Omron CX-Programmer project NewProject (CX-Programmer 9.61)

# PLC NewPLC1: CP1E E20

## Global symbols (name address type ; comment)
0.12 BOOL  ; StopButton
10.00 BOOL  ; Conveyor
0.04 BOOL  ; BothSW
0.03 BOOL  ; BlueSW
0.02 BOOL  ; YellowSW
0.00 BOOL  ; StartButton
0.01 BOOL  ; JobINSen
0.05 BOOL  ; YTHLS
0.06 BOOL  ; BTHLS
0.07 BOOL  ; YTLLS
0.08 BOOL  ; BTLLS
0.09 BOOL  ; JobOUTSen
0.10 BOOL  ; FS1
0.11 BOOL  ; FS2
100.00 BOOL  ; M0
100.01 BOOL  ; M1
100.02 BOOL  ; M2
100.03 BOOL  ; M3
100.04 BOOL  ; M4
100.05 BOOL  ; M5
100.06 BOOL  ; M6
10.01 BOOL  ; YLIndicator
10.02 BOOL  ; BLIndicator
10.03 BOOL  ; YellowValve
10.04 BOOL  ; BlueValve
T000 BOOL  ; Tim1
T001 BOOL  ; Tim2
T002 BOOL  ; Tim3
T003 BOOL  ; Tim4
T004 BOOL  ; Tim5

## Program NewProgram1 (cyclic task 0)

### Section Section1

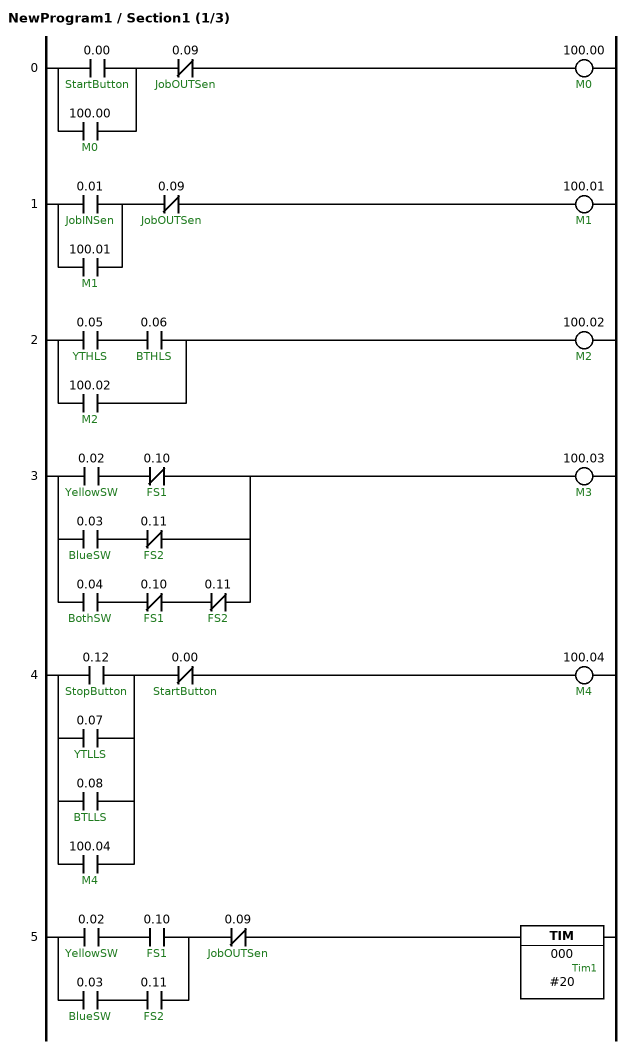
; rung 0
LD 0.00  ; StartButton
OR 100.00  ; M0
ANDNOT 0.09  ; JobOUTSen
OUT 100.00  ; M0
; rung 1
LD 0.01  ; JobINSen
OR 100.01  ; M1
ANDNOT 0.09  ; JobOUTSen
OUT 100.01  ; M1
; rung 2
LD 0.05  ; YTHLS
AND 0.06  ; BTHLS
OR 100.02  ; M2
OUT 100.02  ; M2
; rung 3
LD 0.02  ; YellowSW
ANDNOT 0.10  ; FS1
LD 0.03  ; BlueSW
ANDNOT 0.11  ; FS2
ORLD
LD 0.04  ; BothSW
ANDNOT 0.10  ; FS1
ANDNOT 0.11  ; FS2
ORLD
OUT 100.03  ; M3
; rung 4
LD 0.12  ; StopButton
OR 0.07  ; YTLLS
OR 0.08  ; BTLLS
OR 100.04  ; M4
ANDNOT 0.00  ; StartButton
OUT 100.04  ; M4
; rung 5
LD 0.02  ; YellowSW
AND 0.10  ; FS1
LD 0.03  ; BlueSW
AND 0.11  ; FS2
ORLD
ANDNOT 0.09  ; JobOUTSen
TIM 000 #20  ; Tim1

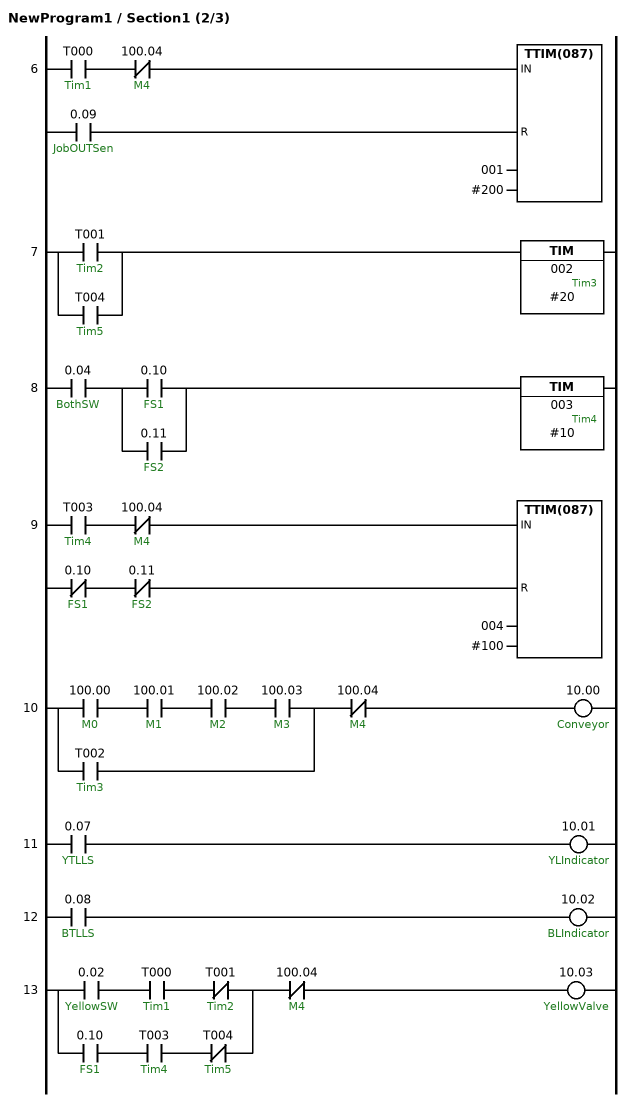
; rung 6
LD T000  ; Tim1
ANDNOT 100.04  ; M4
LD 0.09  ; JobOUTSen
TTIM(087) 001 #200  ; Tim2
; rung 7
LD T001  ; Tim2
OR T004  ; Tim5
TIM 002 #20  ; Tim3
; rung 8
LD 0.04  ; BothSW
LD 0.10  ; FS1
OR 0.11  ; FS2
ANDLD
TIM 003 #10  ; Tim4
; rung 9
LD T003  ; Tim4
ANDNOT 100.04  ; M4
LDNOT 0.10  ; FS1
ANDNOT 0.11  ; FS2
TTIM(087) 004 #100  ; Tim5
; rung 10
LD 100.00  ; M0
AND 100.01  ; M1
AND 100.02  ; M2
AND 100.03  ; M3
OR T002  ; Tim3
ANDNOT 100.04  ; M4
OUT 10.00  ; Conveyor
; rung 11
LD 0.07  ; YTLLS
OUT 10.01  ; YLIndicator
; rung 12
LD 0.08  ; BTLLS
OUT 10.02  ; BLIndicator
; rung 13
LD 0.02  ; YellowSW
AND T000  ; Tim1
ANDNOT T001  ; Tim2
LD 0.10  ; FS1
AND T003  ; Tim4
ANDNOT T004  ; Tim5
ORLD
ANDNOT 100.04  ; M4
OUT 10.03  ; YellowValve

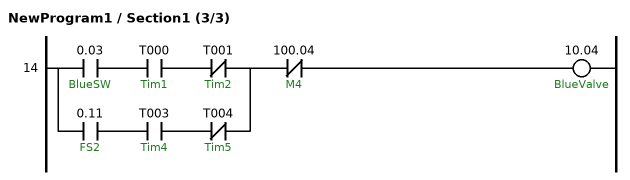
; rung 14
LD 0.03  ; BlueSW
AND T000  ; Tim1
ANDNOT T001  ; Tim2
LD 0.11  ; FS2
AND T003  ; Tim4
ANDNOT T004  ; Tim5
ORLD
ANDNOT 100.04  ; M4
OUT 10.04  ; BlueValve

### Section END
; rung 0
END(001)